(* IEC 61131-3 sources: Daniele1996.github.io/AUTOMATION_AND_SOFTWARE_DESIGN_PATTERN/AUTOMATION_STUDIO/Task2/Logical/Libraries/gAxis_lib, 4 files *)

(* ---- Types.typ ---- *)
TYPE
	gAxis_StateType :
		(
		NotPowered,
		WaitPower,
		Powered,
		Ready,
		CommandHandler,
		MoveVelocity,
		CheckVelocity,
		MoveAdditive,
		CheckPosition,
		CamInState,
		CheckCamState,
		Stop
		);
END_TYPE

(* ---- gAxis.st ---- *)
(* TODO: Add your comment here *)
FUNCTION_BLOCK gAxis

	CASE AxisState OF

		NotPowered:
			IF AxisEnable_in THEN
				gA_Power.Enable := TRUE;
				AxisState := WaitPower;
			END_IF;

		WaitPower:
			IF gA_Power.Status THEN
				gA_Home.Execute := TRUE;
				(*gA_CamTableSelect.Execute := TRUE;*)
				AxisState := Powered;
			END_IF

		Powered:
			(*IF gA_Home.Done AND gA_CamTableSelect.Done THEN*)

			IF gA_Home.Done THEN
				gA_Home.Execute := FALSE;
				AxisEnable_out := FALSE;
				AxisState := Ready;
			END_IF;

		Ready:
			IF AxisCommand = AXIS_MOVE_VELOCITY THEN
				CommandExecuted := FALSE;
				gA_MoveVelocity.Velocity := Velocity;
				gA_MoveVelocity.Execute := TRUE;
				AxisState := MoveVelocity;
			END_IF;

			IF AxisCommand = AXIS_MOVE_ADDITIVE THEN
				CommandExecuted := FALSE;
				gA_MoveAdditive.Distance := Distance;
				gA_MoveAdditive.Execute := TRUE;
				AxisState := MoveAdditive;
			END_IF;

			IF AxisCommand = AXIS_CAM_IN THEN
				CommandExecuted := FALSE;
				gA_CamIn.Execute := TRUE;
				AxisState := CamInState;
			END_IF

			IF AxisCommand = AXIS_STOP THEN
				CommandExecuted := FALSE;
				gA_Stop.Execute := TRUE;
				AxisState := Stop;
			END_IF;

		MoveVelocity:
			IF gA_MoveVelocity.InVelocity THEN
				OldVelocity := Velocity;
				gA_MoveVelocity.Execute := FALSE;
				CommandExecuted := TRUE;
				AxisState := CheckVelocity;
			END_IF;

			IF AxisCommand <> AXIS_MOVE_VELOCITY THEN
				gA_MoveVelocity.Execute := FALSE;
				CommandExecuted := FALSE;
				AxisState := Ready;
			END_IF;

		CheckVelocity:
			IF Velocity <> OldVelocity THEN
				OldVelocity := Velocity;
				gA_MoveVelocity.Velocity := Velocity;
				gA_MoveVelocity.Execute := TRUE;
				CommandExecuted := FALSE;
				AxisState := MoveVelocity;
			END_IF;

			IF AxisCommand <> AXIS_MOVE_VELOCITY THEN
				gA_MoveVelocity.Execute := FALSE;
				CommandExecuted := FALSE;
				AxisState := Ready;
			END_IF;

		MoveAdditive:
			IF gA_MoveAdditive.Done THEN
				OldDistance := Distance;
				gA_MoveAdditive.Execute := FALSE;
				CommandExecuted := TRUE;
				AxisState := CheckPosition;
			END_IF;

			IF AxisCommand <> AXIS_MOVE_ADDITIVE THEN
				gA_MoveAdditive.Execute := FALSE;
				CommandExecuted := FALSE;
				AxisState := Ready;
			END_IF;

		CheckPosition:
			IF Distance <> OldDistance THEN
				OldDistance := Distance;
				gA_MoveAdditive.Distance := Distance;
				gA_MoveAdditive.Execute := TRUE;
				CommandExecuted := FALSE;
				AxisState := MoveAdditive;
			END_IF;

			IF AxisCommand <> AXIS_MOVE_ADDITIVE THEN
				gA_MoveAdditive.Execute := FALSE;
				CommandExecuted := FALSE;
				AxisState := Ready;
			END_IF;

		CamInState:
			IF gA_CamIn.EndOfProfile THEN
				OldCamTableID := CamTableID;
				gA_CamIn.Execute := FALSE;
				CommandExecuted := TRUE;
				AxisState := CheckCamState;
			END_IF

			IF AxisCommand <> AXIS_CAM_IN THEN
				gA_CamIn.Execute := FALSE;
				CommandExecuted := FALSE;
				AxisState :=  Ready;
			END_IF

		CheckCamState:
			IF CamTableID <> OldCamTableID THEN
				OldCamTableID := CamTableID;
				gA_CamIn.Execute := TRUE;
				CommandExecuted := FALSE;
				AxisState := CamInState;
			END_IF;

			IF AxisCommand <> AXIS_MOVE_ADDITIVE THEN
				gA_CamIn.Execute := FALSE;
				CommandExecuted := FALSE;
				AxisState := Ready;
			END_IF;

		Stop:
			IF (gA_Stop.Done) THEN
				CommandExecuted := TRUE;
			END_IF

			IF (AxisCommand <> AXIS_STOP ) THEN
				gA_Stop.Execute := FALSE;
				CommandExecuted := FALSE;

				AxisState := Ready;
			END_IF

	END_CASE;

	AxisEnable_in := AxisEnable_out;

	gA_Power.Axis := Slave;
	gA_Power();

	gA_Home.Axis := Slave;
	gA_Home.Position := Position;
	gA_Home();

	(*
	gA_CamTableSelect.Master := Master;
	gA_CamTableSelect.Slave := Slave;
	gA_CamTableSelect.CamTable := 'Cam';
	gA_CamTableSelect.Periodic := mcNON_PERIODIC;
	gA_CamTableSelect();
	CamTableID := gA_CamTableSelect.CamTableID;
	*)

	gA_MoveVelocity.Axis := Slave;
	gA_MoveVelocity.Velocity := Velocity;
	gA_MoveVelocity.Acceleration := Acceleration;
	gA_MoveVelocity.Deceleration := Deceleration;
	gA_MoveVelocity();

	IF OldDistance = 0 THEN
		OldDistance := Distance;
	END_IF;

	gA_MoveAdditive.Axis := Slave;
	gA_MoveAdditive.Distance := Distance;
	gA_MoveAdditive.Velocity := Velocity;
	gA_MoveAdditive.Acceleration := Acceleration;
	gA_MoveAdditive.Deceleration := Deceleration;
	gA_MoveAdditive();

	gA_ReadActualPosition.Axis := Slave;
	gA_ReadActualPosition.Enable := TRUE;
	gA_ReadActualPosition();

	ActualPosition := gA_ReadActualPosition.Position;

	gA_ReadActualVelocity.Axis := Slave;
	gA_ReadActualVelocity.Enable := TRUE;
	gA_ReadActualVelocity();

	ActualVelocity := gA_ReadActualVelocity.Velocity;

	gA_CamIn.CamTableID := CamTableID;
	gA_CamIn.StartMode := StartMode;
	gA_CamIn.MasterScaling := MasterScaling;
	gA_CamIn.SlaveScaling := SlaveScaling;
	gA_CamIn.MasterOffset := MasterOffset;
	gA_CamIn.SlaveOffset := SlaveOffset;
	gA_CamIn(Master := Master, Slave := Slave);

	gA_CamOut(Slave:=Slave);

	gA_Stop.Axis := Slave;
	gA_Stop.Deceleration := Deceleration;
	gA_Stop();

	gA_ReadStatus.Enable := TRUE;
	gA_ReadStatus.Axis := Slave;
	gA_ReadStatus();

	IF gA_ReadStatus.StandStill THEN
		AxisStatus := STANDSTILL;
	END_IF;

	IF gA_ReadStatus.DiscreteMotion THEN
		AxisStatus := DISCRETE_MOTION;
	END_IF;

	IF gA_ReadStatus.ContinuousMotion THEN
		AxisStatus := CONTINOUS_MOTION;
	END_IF;

END_FUNCTION_BLOCK

(* ---- gAxis_lib.fun ---- *)
FUNCTION_BLOCK gAxis (*TODO: Add your comment here*) (*$GROUP=User,$CAT=User,$GROUPICON=User.png,$CATICON=User.png*)
	VAR_INPUT
		Master : UDINT;
		Slave : UDINT;
		AxisOperation : INT;
		AxisCommand : WORD := 777;
		Distance : REAL;
		Position : REAL;
		Velocity : REAL;
		Acceleration : REAL;
		Deceleration : REAL;
		Jerk : REAL;
		Direction : USINT;
		ArraySize : INT;
		Scale : REAL;
		Offset : REAL;
		RatioNumerator : INT;
		RatioDenominator : INT;
		CamTableID : USINT;
		MasterScaling : REAL := 360;
		SlaveScaling : REAL := 360;
		MasterOffset : REAL := 10;
		SlaveOffset : REAL := 0;
		StartMode : USINT := 1; (*mcRELATIVE*)
		AxisEnable_in : BOOL;
		Reset : BOOL;
	END_VAR
	VAR_OUTPUT
		ActualPosition : REAL;
		ActualVelocity : REAL;
		AxisEnable_out : BOOL;
		CommandExecuted : BOOL := FALSE;
		CommandAborted : BOOL;
		AxisStatus : WORD;
		AxisError : BOOL;
		AxisErrorID : WORD;
		AxisNotInizialized : BOOL;
	END_VAR
	VAR
		INIT : INT;
		RUN : INT;
		OldDistance : REAL;
		OldVelocity : REAL;
		OldCamTableID : USINT;
		AxisState : gAxis_StateType := NotPowered;
		gA_Power : MC_Power;
		gA_Home : MC_Home;
		gA_MoveVelocity : MC_MoveVelocity;
		gA_MoveAdditive : MC_MoveAdditive;
		gA_CamIn : MC_CamIn;
		gA_CamOut : MC_CamOut;
		gA_ReadActualPosition : MC_ReadActualPosition;
		gA_ReadActualVelocity : MC_ReadActualVelocity;
		gA_ReadAxisError : MC_ReadAxisError;
		gA_ReadStatus : MC_ReadStatus;
		gA_Stop : MC_Stop;
	END_VAR
END_FUNCTION_BLOCK

(* ---- Constants.var ---- *)
VAR CONSTANT
	AXIS_NULL_COMMAND : WORD := 0;
	AXIS_MOVE_VELOCITY : WORD := 1;
	AXIS_MOVE_ADDITIVE : WORD := 2;
	AXIS_CAM_IN : WORD := 3;
	AXIS_STOP : WORD := 4;
	STANDSTILL : WORD := 5;
	DISCRETE_MOTION : WORD := 6;
	CONTINOUS_MOTION : WORD := 7;
END_VAR
